Staubli VAL3: SettingCNV.dtx

num nCOLMAX = 39
num nCOLMIN
public num nColumn
public num nFocused
public num nListSize
num nROWMAX = 12
num nROWMIN
public num nRow
string sErrorMessage
string sErrorMsg[10]
  [1] = "An error has been detected in the Page library *\../*"
  [2] = "Variable sTxtBoxLen[*] has an illegal value"
  [3] = "Variable sTxtBoxPos[*] has an illegal value"
  [4] = "The variable *\../* does not exist in the definition library called *\../*"
public string sFALSE = "FALSE"
public string sLabel[4]
  [0] = "-Advanced--"
  [1] = "-Conveyor--"
  [2] = "-TrackingWindow--"
  [3] = "-Event Logger --"
public string sLabelPos[4]
  [0] = "22;0"
  [1] = "0;0"
  [2] = "0;6"
  [3] = "22;7"
public string sListItem0
public string sListItem1
public string sListItem5
public string sListItem6
public string sListItem8
public string sMenu = "; GENERAL ; ENCODER DETECT ; ; Ok"
public string sTRUE = "TRUE"
public string sTitle
public string sTxtBoxAuthord[12]
  [0] = "abcdefghijklmnopqrstuvwxyz_ABCDEFGHIJKLMNOPQRSTUVWXYZ"
  [1] = "abcdefghijklmnopqrstuvwxyz_ABCDEFGHIJKLMNOPQRSTUVWXYZ"
  [2] = "0123456789"
  [3] = "0123456789.-"
  [4] = "0123456789.-"
  [5] = "0123456789."
  [6] = "0123456789."
  [7] = "0123456789."
  [8] = "abcdefghijklmnopqrstuvwxyz_ABCDEFGHIJKLMNOPQRSTUVWXYZ"
  [9] = "0123456789."
  [10] = "0123456789."
  [11] = "abcdefghijklmnopqrstuvwxyz_ABCDEFGHIJKLMNOPQRSTUVWXYZ"
public string sTxtBoxCaption[12]
  [0] = "EncoderLib: "
  [1] = "Detect Lib: "
  [2] = "BufferSize: "
  [3] = "ScaleFact : "
  [4] = "Height    :"
  [5] = "ThruUpLim :"
  [6] = "ThruDwnLim:"
  [7] = "MatchTol: "
  [8] = "ClkSignal:"
  [9] = "ClkPeriod: "
  [10] = "LockDist : "
  [11] = "Enable Log:"
public string sTxtBoxLen[12]
  [0] = "8"
  [1] = "8"
  [2] = "8"
  [3] = "8"
  [4] = "6"
  [5] = "6"
  [6] = "6"
  [7] = "6"
  [8] = "6"
  [9] = "5"
  [10] = "5"
  [11] = "5"
public string sTxtBoxPos[12]
  [0] = "0;1"
  [1] = "0;2"
  [2] = "0;3"
  [3] = "0;4"
  [4] = "0;7"
  [5] = "0;8"
  [6] = "0;9"
  [7] = "22;1"
  [8] = "22;3"
  [9] = "22;4"
  [10] = "22;5"
  [11] = "22;8"
public string sTxtBoxRange[12]
  [2] = "5;200"
  [3] = "-1000;1000"
  [4] = "0;1000"
  [5] = " "
  [6] = " "
  [7] = "1;1000"
  [9] = "0;1000"
  [10] = "0;1000"
public string sTxtBoxType[12]
  [0] = "L1;20;12;5"
  [1] = "L2;20;12;5"
  [2] = "N"
  [3] = "N"
  [4] = "N"
  [5] = "L3;10;12;8"
  [6] = "L4;10;12;8"
  [7] = "N"
  [8] = "L4;18;12;8"
  [9] = "N"
  [10] = "N"
  [11] = "B"
public string sTxtBoxVal[12]
  [0] = "GenericDet"
  [1] = "GenericEnc"
  [2] = "5"
  [3] = "0"
  [4] = "500"
  [7] = "5"
  [9] = "0"
  [10] = "0"
